FUNCTION_BLOCK PUBLIC MotorControl
VAR_INPUT
	CW_Automatic: BOOL;
	CCW_Automatic: BOOL;
	
	
	
	CW_STOP_POS: BOOL;
	CCW_STOP_POS: BOOL;
	
	CURRENT_COUNTROL: INT;
END_VAR
VAR_OUTPUT
END_VAR
VAR
	CW: BOOL;
	CCW: BOOL;
	Direction: BOOL;
END_VAR

//IF CW THEN
//	Direction := TRUE;
//END_IF

//IF CCW THEN
//	Direction := FALSE;
//END_IF

//CW_Timer((),);

END_FUNCTION_BLOCK

(* stored: Version 1.1.0.1, ProductVersion 3.1.4024.13
   POU MotorControl: Id {14ccf3d2-27f3-4cd8-9f85-3d1a66a71ce9}, SpecialFunc None *)
